PROGRAM PRG_SineWave
VAR
    // Sine trajectory
    fTime           : LREAL;                    // Elapsed time [s]
    fCycleTime      : LREAL := 0.001;           // PLC cycle time [s]
    fXRef           : LREAL;                    // Position reference [m]
    fXDotRef        : LREAL;                    // Velocity reference [m/s]
 
    // Feed-forward
    fbFF            : FB_FeedForward_;          // FB for feed-forward
    fbKvFF          : FB_KvFeedForward;         // FB for Kv-based feed-forward
	
    // Position feedback
    fbPosFB         : FB_PositionFeedback;
 
    // Start delay
    fbStartDelay    : TON;
 
    // PF damping
    fbDamping       : FB_PF_Auto;
    ePFMode         : E_PressureFeedback := E_PressureFeedback.PF_ON;
    fDampingGain    : LREAL := 0.0005;
	FilterTime		: LREAL := 0.01;
	fVelocityThr    : LREAL := 0.01;            // Velocity threshold, below this PF will not be active
    bPF_Enabled     : BOOL;                     // Enable signal for PF   
END_VAR

fbStartDelay(IN := G_Inputs.bStartButton AND G_Mode.bRunning AND G_Mode.bAuto, PT := T#2S);

IF fbStartDelay.Q THEN
    fTime := fTime + fCycleTime;
 
    // Sine position reference: x(t) = Mean + A * sin(2*pi*f*t)
    fXRef    := G_Parameter.fMean + G_Parameter.fAmplitude * SIN(2.0 * 3.14159265 * G_Parameter.fFrequency * fTime);
 
    // Velocity reference: x_dot(t) = A * 2*pi*f * cos(2*pi*f*t)
    fXDotRef := G_Parameter.fAmplitude * 2.0 * 3.14159265 * G_Parameter.fFrequency * COS(2.0 * 3.14159265 * G_Parameter.fFrequency * fTime);
 
    G_OPC.fXRef    := fXRef;
    G_OPC.fXDotRef := fXDotRef;
 
    // Feed Forward selection
    CASE G_Enables.eFFMode OF 
		
		 E_FFMode.FF:                              
        	fbFF(
    			bEnable    := G_Enables.bEnableFF,
    			fXDot      := fXDotRef,
    			fPa        := G_OPC.fPaFiltered,
    			fPb        := G_OPC.fPbFiltered,
    			fPs        := G_OPC.fPsFiltered,
    			fA         := G_Parameter.fAreaUp,
    			fAr        := G_Parameter.fAreaDown,
    			fQ0Up      := G_Parameter.fQMaxUp,        
    			fQ0Down    := G_Parameter.fQMaxDown,     
    			fDp0       := G_Parameter.fDeltaP0,       
   				fDeadUp    := G_Parameter.fDeadUp,
    			fDeadDown  := G_Parameter.fDeadDown,
    			fU_FF      => G_OPC.fFF
				);
        
        E_FFMode.KvFF:                              
            fbKvFF(
                bEnable := G_Enables.bEnableFF,
                fXDotref   := fXDotRef,
                fPa     := G_OPC.fPaLowerFiltered,
                fPb     := G_OPC.fPbFiltered,
                fPs     := G_OPC.fPsFiltered,
                fA      := G_Parameter.fAreaUp,
                fAr     := G_Parameter.fAreaDown,
                fU_FF   => G_OPC.fFF
            );
    END_CASE
	
    // Position feedback
    fbPosFB(
        bEnable    := G_Enables.bEnablePositionFeedback,
        fXRef      := fXRef,
        fXActual   := G_OPC.fPistonPosition,
        fKp        := G_Parameter.Kp,
        fKi        := G_Parameter.Ki,
        fKd        := G_Parameter.Kd,
        fCycleTime := fCycleTime,
        fU_PID     => G_OPC.fPID
    );

    G_OPC.fU := G_OPC.fFF + G_OPC.fPID;    // Valve command from FF and position feedback
 
ELSE
    fTime    := 0.0;
    G_OPC.fU := 0.0;
END_IF

// Pressure feedback damping
bPF_Enabled := (ePFMode = E_PressureFeedback.PF_ON) AND (ABS(fXDotRef) > fVelocityThr);	// Controls enable signal according to velocity treshold

fbDamping(
    bEnable := bPF_Enabled,
    fU_In   := G_OPC.fU,
    fKf     := fDampingGain,
    fTauF   := FilterTime,
    fU_Out  => G_OPC.fU
);
 
G_OPC.fU := G_OPC.fU; // Deadband is compensated for in the FF 
 
G_OPC.fU := LIMIT(-1.0, G_OPC.fU, 1.0);    // Safety limit

END_PROGRAM

(* stored: Version 1.1.0.1
   POU PRG_SineWave: Id {0d8dbe2f-c428-4c3a-9aaf-fe8a8124e3c3}, SpecialFunc None *)
